PROGRAM P_Motion
VAR
	fbSineMotionRefMain	: FB_SineMotionRef;
	fbSineMotionRefJib	: FB_SineMotionRef;
	
	fbHomingMainTest	: FB_Homing;
	fbHomingJibTest		: FB_Homing;
	fbHomingWinchTest	: FB_Homing;
	
	fbInitPosMain 		: FB_InitialPos;
	fbInitPosJib		: FB_InitialPos;
	
	fbIntegrator		: FB_Integrator;
END_VAR

fbSineMotionRefMain(
	fInitialPos := fbInitPosMain.fInitialPos
);

fbSineMotionRefJib(
	fInitialPos := fbInitPosJib.fInitialPos
);

fbInitPosMain(
	bEnable := G_Enables.bHoldButton AND G_Enables.bEnableTwo,
	fCurrentPos := G_OPC.fMainPistonPosition.fDanielFilter
);

fbInitPosJib(
	bEnable := G_Enables.bHoldButton AND G_Enables.bEnableOne,
	fCurrentPos := G_OPC.fJibPistonPosition.fDanielFilter
);



IF G_Enables.bSineMotion AND G_Enables.bHoldButton THEN
	fbSineMotionRefMain(
		bEnableMotion := G_Enables.bSineMotion AND G_Enables.bHoldButton AND NOT(G_Enables.bHoming),
		fTime := G_OPC.fMotionTime,
		fFrequency := G_Parameters.fMainFrequency,
		fAmplitude := G_Parameters.fMainAmplitude,
		
		fXDotRef => G_OPC.fXDotRefTwo,
		fXRef => G_OPC.fXRefTwo
	);
	
	fbSineMotionRefJib(
		bEnableMotion := G_Enables.bSineMotion AND G_Enables.bHoldButton AND NOT(G_Enables.bHoming),
		fTime := G_OPC.fMotionTime,
		fFrequency := G_Parameters.fJibFrequency,
		fAmplitude := G_Parameters.fJibAmplitude,
		
		fXDotRef => G_OPC.fXDotRefOne,
		fXRef => G_OPC.fXRefOne
	);
	
ELSIF G_Enables.bHoming AND G_Enables.bHoldButton THEN
	
	IF G_HMI.bHomingMainTest THEN
	
		fbHomingMainTest(
			fWantedPositionMain := 0.5,
			fCurrentPosMain := G_OPC.fMainPistonPosition,
			fWantedPositionJib := 0.5,
			fCurrentPosJib := G_OPC.fJibPistonPosition,
			fClock := G_OPC.fHomingTime,
			bEnableHoming := G_Enables.bHoming,
		
			fXDotRefMain => G_OPC.fXDotRefTwo,
			fXDotRefJib => G_OPC.fXDotRefOne
		);
		
	ELSIF G_HMI.bHomingJibTest THEN
		
		fbHomingJibTest(
			fWantedPositionMain := 0.5,
			fCurrentPosMain := G_OPC.fMainPistonPosition,
			fWantedPositionJib := 0.5,
			fCurrentPosJib := G_OPC.fJibPistonPosition,
			fClock := G_OPC.fHomingTime,
			bEnableHoming := G_Enables.bHoming,
		
			fXDotRefMain => G_OPC.fXDotRefTwo,
			fXDotRefJib => G_OPC.fXDotRefOne
		);
		
	ELSIF G_HMI.bHomingWinchTest THEN
		
		fbHomingWinchTest(
			fWantedPositionMain := 0.5,
			fCurrentPosMain := G_OPC.fMainPistonPosition,
			fWantedPositionJib := 0.5,
			fCurrentPosJib := G_OPC.fJibPistonPosition,
			fClock := G_OPC.fHomingTime,
			bEnableHoming := G_Enables.bHoming,
		
			fXDotRefMain => G_OPC.fXDotRefTwo,
			fXDotRefJib => G_OPC.fXDotRefOne
		);
	END_IF
	
ELSE
	
	G_OPC.fXDotRefOne := 0.0;
	G_OPC.fXRefOne := G_OPC.fJibPistonPosition.fDanielFilter;
	
	G_OPC.fXDotRefTwo := 0.0;
	G_OPC.fXRefTwo := G_OPC.fMainPistonPosition.fDanielFilter;
	
END_IF

END_PROGRAM

(* stored: Version 1.1.0.1
   POU P_Motion: Id {e2f87671-7351-4a5e-baec-94080915a986}, SpecialFunc None *)
